{attribute 'linkalways'} 
{attribute 'no_explicit_call' := 'This FB is a CLASS and must be accessed using methods or properties'}
{attribute 'enable_dynamic_creation'}
FUNCTION_BLOCK _ETcVnDistanceTransformationLabel EXTENDS EnumDatatypeBase
VAR
	localData : ETcVnDistanceTransformationLabel;
	activeData : REFERENCE TO ETcVnDistanceTransformationLabel;
	enumBaseDatatype : _DINT(localData);
END_VAR

METHOD PRIVATE AddLocalEnumeration
VAR_INPUT
	Enumeration : T_MAXSTRING;
	Value : ETcVnDistanceTransformationLabel;
END_VAR
AddEnumeration(Enumeration, Value);
END_METHOD

PROPERTY PUBLIC Address : PVOID
GET
Address := ADR(activeData);
END_GET
END_PROPERTY

METHOD PUBLIC ClearReference
VAR_INPUT
END_VAR
activeData REF= localData;
SetBaseDatatypeReference();
END_METHOD

METHOD PUBLIC Clone : I_Datatype
VAR
    pClone : POINTER TO _ETcVnDistanceTransformationLabel;
END_VAR
pClone := __NEW(_ETcVnDistanceTransformationLabel(InitialValue := Value));
Clone := pClone^;
END_METHOD

METHOD FB_init : BOOL
VAR_INPUT
	bInitRetains : BOOL; // if TRUE, the retain variables are initialized (warm start / cold start)
	bInCopyCode : BOOL;  // if TRUE, the instance afterwards gets moved into the copy code (online change)
	InitialValue : ETcVnDistanceTransformationLabel;
END_VAR
localData := InitialValue;
AddBaseDatatype(enumBaseDatatype);
ClearReference();

AddLocalEnumeration('TCVN_DTL_CCOMP', ETcVnDistanceTransformationLabel.TCVN_DTL_CCOMP);
AddLocalEnumeration('TCVN_DTL_PIXEL', ETcVnDistanceTransformationLabel.TCVN_DTL_PIXEL);
END_METHOD

PROPERTY PUBLIC Identifier : T_MAXSTRING
GET
Identifier := 'ETcVnDistanceTransformationLabel';
END_GET
END_PROPERTY

METHOD IsEnumeratorValueEqual : BOOL
VAR_INPUT
	Enumerator : I_KeyValueForwardEnumerator;
END_VAR
VAR
	storedValue : ETcVnDistanceTransformationLabel;
END_VAR
IF NOT Enumerator.TryGet(storedValue) THEN
	RETURN;
END_IF

IsEnumeratorValueEqual := storedValue = activeData;
END_METHOD

METHOD PUBLIC MakeReferenceTo
VAR_INPUT
	ReferenceTarget : REFERENCE TO ETcVnDistanceTransformationLabel;
END_VAR
activeData REF= ReferenceTarget;
SetBaseDatatypeReference();
END_METHOD

METHOD PROTECTED SetBaseDatatypeReference
VAR_INPUT
END_VAR
enumBaseDatatype.MakeReferenceTo(activeData);
END_METHOD

PROPERTY PUBLIC Size : UDINT
GET
Size := SIZEOF(activeData);
END_GET
END_PROPERTY

METHOD TryMakeReferenceTo : BOOL
VAR_INPUT
	Target : I_Datatype;
END_VAR
VAR
	pTargetData : POINTER TO ETcVnDistanceTransformationLabel;
END_VAR
IF NOT IsEquivalentTo(Target) THEN
	RETURN;
END_IF

pTargetData := Target.Address;
activeData REF= pTargetData^;
SetBaseDatatypeReference();
TryMakeReferenceTo := TRUE;
END_METHOD

PROPERTY PUBLIC Value : ETcVnDistanceTransformationLabel
GET
Value := activeData;
END_GET
SET
activeData := Value;
END_SET
END_PROPERTY

END_FUNCTION_BLOCK

(* stored: Version 1.1.0.1, ProductVersion 3.1.4024.13
   POU _ETcVnDistanceTransformationLabel: Id {19a31a00-f7de-062c-3c2e-b4f2cd0a662b}, SpecialFunc None
   Folder Core: Id {768fddc6-bae8-0a5b-3b80-63b1c26ffd24}
   Folder Protected: Id {d303fd09-e94a-0e7e-2921-5d6bb8d01397}
   Folder Customize: Id {56192f5c-b0a0-0fea-275e-1ac832ed0f48}
   Folder Constructor: Id {dd891b2d-8fcb-0fa0-012b-7c190d8fa942}
   Folder Private: Id {7e180948-85f2-0950-0264-9abf534b59ce}
   Folder Protected: Id {a86a076c-bca3-0c58-378e-5f7804072df8}
   Method AddLocalEnumeration: Id {e4897d57-4c5a-0cbb-2502-5f08e8f7a6f2}
   Property Address: Id {252c366c-1aff-0531-086c-3984235a4d4b}
   Get Get: Id {7a911c27-8645-0438-0593-e7619064608a}
   Method ClearReference: Id {e12ffe52-d342-0c2a-38ca-04405644a653}
   Method Clone: Id {85af352d-fef7-0ef2-3a3a-b5d4b0f55867}
   Method FB_init: Id {dbc87442-f00e-0193-39d2-45e5645caf1b}
   Property Identifier: Id {06676978-8db0-0e34-1534-15ce1d3627ab}
   Get Get: Id {4e3b9b1b-48d0-0d67-0288-203b1716860e}
   Method IsEnumeratorValueEqual: Id {5f2baf6d-8ee3-0c6d-1f8f-0f00b9e159de}
   Method MakeReferenceTo: Id {39be66e3-d534-0fc2-286c-3b822cc09f2a}
   Method SetBaseDatatypeReference: Id {f1c380e3-74db-07fd-0b46-040aa6199d1d}
   Property Size: Id {3683bbc9-749c-0b65-1c8c-b5383c66e9fb}
   Get Get: Id {b53204e6-c872-0a58-1ea7-f3b2e63e6ef0}
   Method TryMakeReferenceTo: Id {b2bdbac6-cba6-0a37-26b9-edeb7eb28f43}
   Property Value: Id {36876ed5-9b55-0b10-25eb-10c5b65691a4}
   Get Get: Id {d3c7388a-2986-0248-04a6-0c710c6925b3}
   Set Set: Id {5c537a1c-a4a6-037d-3301-39e6a52f35d4} *)
